# EPICS SNL sequencer program: zfhifiSup/zero_field.st
program zero_field("P")

#include "ibexSeqPVmacros.h"
#include "zf_pv_definitions.h"
%% #include "seq_snc.h"
%% #include "epicsTime.h"
%% #include "string.h"
%% #include "math.h"
%% #include "errlog.h"
%% #include "alarm.h"

option +d;
option +r;
option +s;

%{
  static const char* const PROGRAM_NAME = "zero_field.st";

  /* Define some error statuses. These should match the indices in $(P)STATUS */
  static const int ZF_STAT_NO_ERROR = 0;
  static const int ZF_STAT_MAGNETOMETER_DATA_STALE = 1;
  static const int ZF_STAT_MAGNETOMETER_DATA_INVALID = 2;
  static const int ZF_STAT_MAGNETOMETER_DATA_INVALID_MANUAL = 3;
  static const int ZF_STAT_PSU_INVALID = 4;
  static const int ZF_STAT_PSU_ON_LIMITS = 5;
  static const int ZF_STAT_PSU_WRITE_FAILED = 6;
  static const int ZF_STAT_PSU_LIMITS_INCONSISTENT = 7;
  static const int ZF_STAT_PSU_SP_RBV_OUT_OF_RANGE = 8;

  static const int PSU_STATUS_OFF = 0;
  static const int PSU_STATUS_ON = 1;

  /* This needs to be a macro as the call to pvIndex has to happen from SNL code, not C code. */
  /* See https://www-csr.bessy.de/control/SoftDist/sequencer/EscapeToC.html?highlight=pvindex#calling-pv-functions-from-c */
  #define ZF_TRANSITION_TO_STATE(x) zf_state_transition(ssId, pVar, pvIndex(statemachine_state), (x))

  /* Some necessary function forward-declarations - for implementations see end of file. */
  static void zf_state_transition(SS_ID ssId, struct seqg_vars* const pVar, CH_ID index, const char* const new_state_name);
  static int power_supplies_invalid(struct seqg_vars* const pVar);
  static int magnetometer_invalid(struct seqg_vars* const pVar);
  static int is_within_tolerance(double setpoint, double readback, double tolerance);
  static void report_tolerance_error(const char* axis, double sp, double sp_rpv, double tolerance, double timeout);
  static double coerce_to_range(double value, double low_limit, double high_limit);
  static int psu_sp_rbv_out_of_range(struct seqg_vars* const pVar);

  /* A timestamp from the last time we asked the magnetometer to take data. Used for loop time calculation. */
  epicsTimeStamp _time_of_last_mag_read_trigger;
  epicsTimeStamp _time_of_last_psu_write_trigger;
  epicsTimeStamp _time_of_last_psu_check_trigger;

  /* flag to track whether power supply outputs were limited or not. Need this flag to be able to set correct errors. */
  int _output_on_limit = 0;
}%

ss zero_field
{

  /* Initial state. */
  state initializing
  {
    entry {
      ZF_TRANSITION_TO_STATE("initializing");
      %% epicsTimeGetCurrent(&_time_of_last_mag_read_trigger);
	  statemachine_activity = 0;
    }
    when (){} state trigger_mag_read
  }

  state trigger_mag_read
  {
    entry {
      %% epicsTimeStamp new_time;
      %% double time_taken;
      ZF_TRANSITION_TO_STATE("trigger_mag_read");

      /* inverts each time around the main statemachine loop, giving a flashing effect if everything is working correctly. */
      PVPUT(statemachine_activity, !statemachine_activity);
      %% epicsTimeGetCurrent(&new_time);
      %% time_taken = 1000.0 * epicsTimeDiffInSeconds(&new_time, &_time_of_last_mag_read_trigger);
      PVPUT(statemachine_measured_loop_time, time_taken);

      if (debug) {
        errlogSevPrintf(errlogInfo, "%s: Loop took %f ms.\n", PROGRAM_NAME, time_taken);
      }

      _time_of_last_mag_read_trigger = new_time;
      PVPUTF(readings_ready_set, 0, SYNC);
    }

    when(!readings_ready) {
      PVPUT(trigger_readings, 1);
    } state wait_for_mag_read
  }

  state wait_for_mag_read
  {
    entry {
      ZF_TRANSITION_TO_STATE("wait_for_mag_read");
    }

    when(
	  readings_ready && !magnetometer_invalid(pVar)
	) {
      %% epicsTimeStamp new_time;
      %% double time_taken;
     /* make sure we definitely have readings */
	  pvGet(magnetometer_x, SYNC);
	  pvGet(magnetometer_y, SYNC);
	  pvGet(magnetometer_z, SYNC);
      %% epicsTimeGetCurrent(&new_time);
      %% time_taken = 1000.0 * epicsTimeDiffInSeconds(&new_time, &_time_of_last_mag_read_trigger);
	  PVPUT(statemachine_measured_read_time, time_taken);
    } state check_corrected_field

    when(
	  readings_ready && magnetometer_invalid(pVar)
	) {
      %% epicsTimeStamp new_time;
      %% double time_taken;
      if (auto_feedback_enabled) {
        PVPUT(at_setpoint, 0);
      }
      PVPUT(status,  auto_feedback_enabled ? ZF_STAT_MAGNETOMETER_DATA_INVALID : ZF_STAT_MAGNETOMETER_DATA_INVALID_MANUAL);
      errlogSevPrintf(errlogMajor, "%s: Magnetometer read error: new reading became available but severities were invalid.\n", PROGRAM_NAME);
      %% epicsTimeGetCurrent(&new_time);
      %% time_taken = 1000.0 * epicsTimeDiffInSeconds(&new_time, &_time_of_last_mag_read_trigger);
      PVPUT(statemachine_measured_read_time, time_taken);
    } state wait_before_read

    when(delay(read_timeout)) {
      if (auto_feedback_enabled) {
        PVPUT(at_setpoint, 0);
      }
	  PVPUT(statemachine_measured_read_time, read_timeout * 1000.0);
      PVPUT(status, ZF_STAT_MAGNETOMETER_DATA_STALE);
      errlogSevPrintf(errlogMajor, "%s: Magnetometer read error: new reading did not become available.\n", PROGRAM_NAME);
    } state trigger_mag_read
  }

  state check_corrected_field {
    entry {
      ZF_TRANSITION_TO_STATE("check_corrected_field");
    }

    when(delay(0.1)) {  /* TOM TODO: make this configurable */
      if (!auto_feedback_enabled) {
        PVPUT(at_setpoint, 2);
      } else {
        int within_tolerance = is_within_tolerance(setpoint_x, magnetometer_x, tolerance) &&
            is_within_tolerance(setpoint_y, magnetometer_y, tolerance) &&
            is_within_tolerance(setpoint_z, magnetometer_z, tolerance);

        PVPUT(at_setpoint, within_tolerance);

        if (debug) {
          errlogSevPrintf(errlogInfo, "%s: Magnetometer within tolerance: %s\n", PROGRAM_NAME, within_tolerance ? "True" : "False");
        }
      }
    } state check_auto_feedback
  }

  state check_auto_feedback {
    entry {
      ZF_TRANSITION_TO_STATE("check_auto_feedback");
    }

    when(auto_feedback_enabled) {
      /* Intentionally empty */
    } state check_output_psu_state

    when(!auto_feedback_enabled) {
      /* If we get to this point, there is no error. Clear any previous error states. */
      PVPUT(status, ZF_STAT_NO_ERROR);

      if (debug) {
        errlogSevPrintf(errlogMajor, "%s: Auto-feedback disabled - skipping PSU writes\n", PROGRAM_NAME);
      }
    } state wait_before_read
  }

  state check_output_psu_state {
    entry {
      ZF_TRANSITION_TO_STATE("check_output_psu_state");
    }

    when(power_supplies_invalid(pVar)) {
      PVPUT(status, ZF_STAT_PSU_INVALID);
      errlogSevPrintf(errlogMajor, "%s: Power supply is in invalid alarm. Not writing to power supplies.\n", PROGRAM_NAME);
    } state wait_before_read

    when(!power_supplies_invalid(pVar)) {
      /* Intentionally empty */
    } state write_to_psu
  }

  state write_to_psu {
    entry {
      ZF_TRANSITION_TO_STATE("write_to_psu");
      %% epicsTimeGetCurrent(&_time_of_last_psu_write_trigger);
    }

    when() {
     /* make sure we definitely have readings */
      %% epicsTimeStamp new_time;
      %% double time_taken;
      double new_x, new_y, new_z, coerced_x, coerced_y, coerced_z;
	  int x_on_limit, y_on_limit, z_on_limit;

      new_x = output_psu_x + (setpoint_x - magnetometer_x) * feedback;
      new_y = output_psu_y + (setpoint_y - magnetometer_y) * feedback;
      new_z = output_psu_z + (setpoint_z - magnetometer_z) * feedback;

      coerced_x = coerce_to_range(new_x, output_psu_x_sp_drvl, output_psu_x_sp_drvh);
      coerced_y = coerce_to_range(new_y, output_psu_y_sp_drvl, output_psu_y_sp_drvh);
      coerced_z = coerce_to_range(new_z, output_psu_z_sp_drvl, output_psu_z_sp_drvh);

      x_on_limit = (new_x != coerced_x);
      y_on_limit = (new_y != coerced_y);
      z_on_limit = (new_z != coerced_z);

      if (x_on_limit || y_on_limit || z_on_limit) {
        errlogSevPrintf(errlogMajor, "%s: power supply outputs on limits. Attempted to set (X=%f, Y=%f, Z=%f) but instead set (X=%f, Y=%f, Z=%f)\n",
          PROGRAM_NAME, new_x, new_y, new_z, coerced_x, coerced_y, coerced_z);

        /* error set in check_psu_writes based on this flag */
        _output_on_limit = 1;
      } else {
        _output_on_limit = 0;
      }

      if (debug) {
        errlogSevPrintf(errlogInfo, "%s: Writing to power supplies X=%f, Y=%f, Z=%f",
		                PROGRAM_NAME, coerced_x, coerced_y, coerced_z);
      }

      PVPUT(output_psu_x_sp, coerced_x);
      PVPUT(output_psu_y_sp, coerced_y);
      PVPUT(output_psu_z_sp, coerced_z);

	  %% epicsTimeGetCurrent(&new_time);
      %% time_taken = 1000.0 * epicsTimeDiffInSeconds(&new_time, &_time_of_last_psu_write_trigger);
	  PVPUT(statemachine_measured_write_time, time_taken);

    } state check_psu_writes
  }

  state check_psu_writes {
      entry {
        ZF_TRANSITION_TO_STATE("check_psu_writes");
        %% epicsTimeGetCurrent(&_time_of_last_psu_check_trigger);
      }

      when(
        is_within_tolerance(output_psu_x_sp, output_psu_x, output_psu_tolerance) &&
        is_within_tolerance(output_psu_y_sp, output_psu_y, output_psu_tolerance) &&
        is_within_tolerance(output_psu_z_sp, output_psu_z, output_psu_tolerance) &&
		output_psu_x_ready &&
		output_psu_y_ready &&
		output_psu_z_ready
      ) {
        %% epicsTimeStamp new_time;
        %% double time_taken;
        if (_output_on_limit) {
          PVPUT(status, ZF_STAT_PSU_ON_LIMITS);
        } else {
          /* If we get to this state, there has been no error */
          PVPUT(status, ZF_STAT_NO_ERROR);
        }

        if (debug) {
          errlogSevPrintf(errlogInfo, "%s: power supply writes successful X=%f, Y=%f, Z=%f\n",
		                  PROGRAM_NAME, output_psu_x, output_psu_y, output_psu_z);
        }
		%% epicsTimeGetCurrent(&new_time);
        %% time_taken = 1000.0 * epicsTimeDiffInSeconds(&new_time, &_time_of_last_psu_check_trigger);
	    PVPUT(statemachine_measured_check_time, time_taken);
      } state wait_before_read

      when(delay(write_timeout)) {
          PVPUT(status, ZF_STAT_PSU_WRITE_FAILED);
		  report_tolerance_error("X", output_psu_x_sp, output_psu_x, output_psu_tolerance, write_timeout);
		  report_tolerance_error("Y", output_psu_y_sp, output_psu_y, output_psu_tolerance, write_timeout);
		  report_tolerance_error("Z", output_psu_z_sp, output_psu_z, output_psu_tolerance, write_timeout);
	      PVPUT(statemachine_measured_check_time, write_timeout * 1000.0);

       /*do not go to wait_before_read in this case as we have already waited for write_timeout */
      } state trigger_mag_read
  }

  state wait_before_read {
    entry {
      ZF_TRANSITION_TO_STATE("wait_before_read");
    }

    when(delay(loop_delay/1000.0)) { } state trigger_mag_read
  }
}

%{
  /**
   * Called on any state transitions that occur in the state machine - primarily for debugging.
   */
  static void zf_state_transition(SS_ID ssId, struct seqg_vars* const pVar, CH_ID index, const char* const new_state_name)
  {
    strncpy(pVar->statemachine_state, new_state_name, MAX_STRING_SIZE);
	seq_pvPut(ssId, index, SYNC);
    if (pVar->debug) {
	  errlogSevPrintf(errlogInfo, "%s: Entering state %s\n", PROGRAM_NAME, new_state_name);
    }
  }

  /**
   * Return 1 if any of the power supply readbacks or setpoint readbacks are invalid - else return 0.
   */
  static int power_supplies_invalid(struct seqg_vars* const pVar) {
    return pVar->output_psu_x_sevr == INVALID_ALARM
        || pVar->output_psu_y_sevr == INVALID_ALARM
        || pVar->output_psu_z_sevr == INVALID_ALARM;
  }

  /**
   * Return 1 if any of the magnetometer readbacks are invalid - else return 0.
   */
  static int magnetometer_invalid(struct seqg_vars* const pVar) {
    return pVar->magnetometer_x_sevr == INVALID_ALARM
        || pVar->magnetometer_y_sevr == INVALID_ALARM
        || pVar->magnetometer_z_sevr == INVALID_ALARM;
  }

  /**
   * Returns 1 if the first two arguments are within tolerance of each other, else 0.
   */
  static int is_within_tolerance(double setpoint, double readback, double tolerance) {
    return fabs(setpoint - readback) <= tolerance;
  }

  /**
   * Report error if axis out of tolerance
   */
    static void report_tolerance_error(const char* axis, double sp, double sp_rbv, double tolerance, double timeout)
    {
        if (!is_within_tolerance(sp, sp_rbv, tolerance)) {
            errlogSevPrintf(errlogMajor, "%s: %s Power supply write failed to get within tolerance %f: SP=%f SP:RBV=%f error=%f Timeout=%f\n",
                          PROGRAM_NAME, axis, tolerance, sp, sp_rbv, sp - sp_rbv, timeout);
        }
    }

  /**
   * Coerces a floating point number to be within given low and high limits.
   */
  static double coerce_to_range(double value, double low_limit, double high_limit) {
    if (high_limit < low_limit) {
      errlogSevPrintf(errlogMajor, "%s: coerce_to_range called with high < low. Returning zero.", PROGRAM_NAME);
      return 0.0;
    }

    if (value > high_limit) {
        return high_limit;
    } else if (value < low_limit) {
        return low_limit;
    } else {
        return value;
    }
  }
}%
